// TIA Portal V20 export
FUNCTION_BLOCK "FB_GetTextErrorCode"   // FB301, SCL
{ S7_Optimized_Access := 'TRUE' }
// stored: AutoNumber false, MemoryReserve 100, SetENOAutomatically false
   VAR_INPUT
      iErrorCode { ExternalAccessible := 'False'; ExternalVisible := 'False'; ExternalWritable := 'False'} : Int;
   END_VAR
   VAR_OUTPUT
      oErrorText { ExternalAccessible := 'False'; ExternalVisible := 'False'; ExternalWritable := 'False'} : String;
   END_VAR
   VAR RETAIN
      sCode_error : Array[0..100] of Struct
         ErrorCode : Int;
         ErrorText : String[64];
      END_STRUCT;
   END_VAR
   VAR_TEMP
      tIndex : Int;
   END_VAR
   // sCode_error[0].ErrorCode := 0;
   // sCode_error[1].ErrorCode := 9999;
   // sCode_error[2].ErrorCode := 7504;
   // sCode_error[3].ErrorCode := 8000;
   // sCode_error[4].ErrorCode := 7064;
   // sCode_error[5].ErrorCode := 7004;
   // sCode_error[6].ErrorCode := 27564;
   // sCode_error[7].ErrorCode := 7068;
   // sCode_error[8].ErrorCode := 17504;
   // sCode_error[9].ErrorCode := 6564;
   // sCode_error[10].ErrorCode := 9064;
   // sCode_error[11].ErrorCode := 9004;
   // sCode_error[12].ErrorCode := 9010;
   // sCode_error[13..100].ErrorCode := 0;
   // sCode_error[0].ErrorText := 'Unknown, No text';
   // sCode_error[1].ErrorText := 'Part start drilling, but not finished';
   // sCode_error[2].ErrorText := 'woz out of tolerance';
   // sCode_error[3].ErrorText := 'runout';
   // sCode_error[4].ErrorText := 'Z out of range';
   // sCode_error[5].ErrorText := 'Z out of tolerance';
   // sCode_error[6].ErrorText := 'woz out of range';
   // sCode_error[7].ErrorText := 'z out of range and tolerance';
   // sCode_error[8].ErrorText := 'part not clamped';
   // sCode_error[9].ErrorText := 'Woc';
   // sCode_error[10..11].ErrorText := 'Drilled part with broken BW';
   // sCode_error[12].ErrorText := 'Drilled part with N2 not enough';
   // sCode_error[13..100].ErrorText := '';
BEGIN
       //==================================================================================
       // POSALUX Swiss SA / (C) Copyright 2025
       //----------------------------------------------------------------------------------
       // Title: Power de la machine
       // Comment/Function: Generates an error text based on an error number
       //           If the Error code is not found, "ErrorCode: Code unknow" is displayed          
       // Author: Fabien WALDT
       // Engineering: TIA Portal v17
       //----------------------------------------------------------------------------------
       // Change log table:
       // Version  | Date     | Expert in charge | Changes applied
       // ---------|----------|------------------|------------------------------------
       // 00.00.01 | 20250415 | WFA              | First released version
       // ==================================================================================
       REGION NO Error
           IF #iErrorCode = 0 THEN
               #oErrorText := #sCode_error[0].ErrorText;
           END_IF;
       END_REGION

       REGION Error
           IF #iErrorCode > 0 THEN
               FOR #tIndex := 1 TO 100 DO
                   IF #iErrorCode = #sCode_error[#tIndex].ErrorCode THEN
                       // Error text found in the list
                       #oErrorText := #sCode_error[#tIndex].ErrorText;
                       EXIT;
                   END_IF;
                   // Error text not found in the list
                   #oErrorText := CONCAT(IN1 := DELETE(IN := INT_TO_STRING(#iErrorCode), L := 1, P := 1), IN2 := ': Code unknow');
               END_FOR;
           END_IF;
       END_REGION
END_FUNCTION_BLOCK
